ORGANIZATION_BLOCK "Main_MES"
TITLE = "Main Program Sweep (Cycle)"
{ S7_Optimized_Access := 'TRUE' ; Published := 'FALSE' }
VERSION : 0.1

BEGIN
	"Production_CALL"();


	"MES_Manager_Call"();


	"IPC_Manager_CALL"();


	"Production_ITF"();

END_ORGANIZATION_BLOCK

